// TIA Portal V17 export
// export: Created 2022-07-20T06:59:44.809316Z, ExportSetting WithDefaults, DisplayName Totally Integrated Automation Portal, DisplayVersion V17, DisplayName TIA Portal Openness, DisplayVersion V17, DisplayName TIA Portal Version Control Interface, DisplayVersion V17, DisplayName SINAMICS Startdrive Advanced, DisplayVersion V17, DisplayName SINAMICS Startdrive G130, G150, S120, S150, SINAMICS MV, S210, DisplayVersion V17, DisplayName SINAMICS Startdrive G110M, G120, G120C, G120D, G120P, G115D, DisplayVersion V17, DisplayName STEP 7 Professional, DisplayVersion V17, DisplayName STEP 7 Safety, DisplayVersion V17, DisplayName WinCC Advanced, DisplayVersion V17
FUNCTION_BLOCK "FB10078_AirExtractorManager_1"   // FB10078, LAD
TITLE = FB10078_AirExtractorManager_1
{ S7_Optimized_Access := 'TRUE' }
AUTHOR : Anirouddh
FAMILY : 1007x_DRYER_UV
VERSION : 1.0
// Release note : 
// 1.0 - Feature improved
// stored: AutoNumber false, IsIECCheckEnabled false, IsRetainMemResEnabled false, MemoryReserve 100, SetENOAutomatically false, UDAEnableTagReadback false
   VAR_INPUT
      UvLampReady : Bool;
      UvLampError : Bool;
      RequestAirExtraction { ExternalAccessible := 'False'; ExternalVisible := 'False'; ExternalWritable := 'False'} : Bool;
      RequestShutDown : Bool;
      ScalingShutterOpen : "stAirExtractorScalingParameters";
      ScalingShutterClosed : "stAirExtractorScalingParameters";
      UVAnalogicalFeedbackPower : Int;
      UVModbusRtuFeedbackPower : UInt;
      ShutterOpen : Bool;
      ShutterClose : Bool;
      PWM_MinFrequenceValue : Real;
      PWM_MaxFrequenceValue : Real;
   END_VAR
   VAR_OUTPUT
      PWM_ActiveAirExtractor : Bool;
      PWM_FrequencyValue : Real;
      Analog_PowerValue : Int;
      ShutDownInProgress : Bool;
      ShutDownDone : Bool;
      ShutDownTime : Time;
   END_VAR
   VAR
      VoltageFeedback_Temp : Real;
      R_TRIG_RequestShutDown { S7_SetPoint := 'True'} : R_TRIG;
      TON_ShutdownTimer { S7_SetPoint := 'True'} : TON_TIME;
   END_VAR
BEGIN

REGION Network 1 (SCL): Edge Signals & Timers
   REGION EDGE SIGNALS
       #R_TRIG_RequestShutDown(CLK := #RequestShutDown);
   END_REGION

   REGION TIMERS
       //Shutdown timer
       #TON_ShutdownTimer(IN := #ShutDownInProgress,
                          PT := T#5m,
                          ET => #ShutDownTime);
   END_REGION
END_REGION

REGION Network 2 (SCL): Air Extractor Management
   //Determine The Feedback Volatge Of The Lamp
   IF #UVAnalogicalFeedbackPower = 0 AND #UVModbusRtuFeedbackPower <> 0 THEN
       #VoltageFeedback_Temp := UINT_TO_REAL(#UVModbusRtuFeedbackPower);
   ELSIF #UVAnalogicalFeedbackPower <> 0 AND #UVModbusRtuFeedbackPower = 0 THEN
       #VoltageFeedback_Temp := #UVAnalogicalFeedbackPower;
   ELSE
       #VoltageFeedback_Temp := #ScalingShutterOpen.PowerXMax;
   END_IF;

   //Determine the Air Extractor Set Point
   IF #RequestAirExtraction AND NOT (#ShutDownInProgress) THEN
       #PWM_ActiveAirExtractor := TRUE;
       IF #ShutterClose THEN
           "FC10072_ScalingAirExtraction_VolatgeFeedback"(VoltageFeedback := #VoltageFeedback_Temp,
                                                          X_UVPower_Min := #ScalingShutterClosed.PowerXMin,
                                                          X_UVPower_Max := #ScalingShutterClosed.PowerXMax,
                                                          Y_AirPower_Min := #ScalingShutterClosed.PowerAirYMin,
                                                          Y_AirPower_Max := #ScalingShutterClosed.PowerAirYMax,
                                                          PWM_Minimum := #PWM_MinFrequenceValue,
                                                          PWM_Maximum := #PWM_MaxFrequenceValue,
                                                          Analogical_Value => #Analog_PowerValue,
                                                          PWM_FrequenceValue => #PWM_FrequencyValue);
       ELSIF #ShutterOpen THEN
           "FC10072_ScalingAirExtraction_VolatgeFeedback"(VoltageFeedback := #VoltageFeedback_Temp,
                                                          X_UVPower_Min := #ScalingShutterOpen.PowerXMin,
                                                          X_UVPower_Max := #ScalingShutterOpen.PowerXMax,
                                                          Y_AirPower_Min := #ScalingShutterOpen.PowerAirYMin,
                                                          Y_AirPower_Max := #ScalingShutterOpen.PowerAirYMax,
                                                          PWM_Minimum := #PWM_MinFrequenceValue,
                                                          PWM_Maximum := #PWM_MaxFrequenceValue,
                                                          Analogical_Value => #Analog_PowerValue,
                                                          PWM_FrequenceValue => #PWM_FrequencyValue);
       END_IF;
   ELSIF #ShutDownInProgress THEN
       #PWM_ActiveAirExtractor := TRUE;
       "FC10072_ScalingAirExtraction_VolatgeFeedback"(VoltageFeedback := #ScalingShutterClosed.PowerXMax,
                                                      X_UVPower_Min := #ScalingShutterClosed.PowerXMin,
                                                      X_UVPower_Max := #ScalingShutterClosed.PowerXMax,
                                                      Y_AirPower_Min := #ScalingShutterClosed.PowerAirYMin,
                                                      Y_AirPower_Max := #ScalingShutterClosed.PowerAirYMax,
                                                      PWM_Minimum := #PWM_MinFrequenceValue,
                                                      PWM_Maximum := #PWM_MaxFrequenceValue,
                                                      Analogical_Value => #Analog_PowerValue,
                                                      PWM_FrequenceValue => #PWM_FrequencyValue);
   ELSE
       #PWM_ActiveAirExtractor := FALSE;
       #PWM_FrequencyValue := 0;
       #Analog_PowerValue := 0;
   END_IF;

   //Air Extractor Shutdown Management
   IF #R_TRIG_RequestShutDown.Q THEN
       #ShutDownInProgress := TRUE;
   ELSIF #TON_ShutdownTimer.Q THEN
       #ShutDownInProgress := FALSE;
       #ShutDownDone := TRUE;
   ELSE
       #ShutDownDone := FALSE;
   END_IF;
END_REGION
END_FUNCTION_BLOCK
